Staubli VAL3: decode.pgx

public program decode(num& x_nStatus (dimensions=1), num& x_nDWordBody[] (dimensions=2))
  local num l_nBodyDWordLen
  local num i
begin
  // x_nStatus
  // -1 - unsuccessful
  // 0 - successful
  x_nStatus=-1
  l_nBodyDWordLen=34
  if size(x_nDWordBody,1)!=l_nBodyDWordLen or size(x_nDWordBody,2)!=4
    put("Size of the param is: "+toString("",size(x_nDWordBody,1)))
    putln("x"+toString("",size(x_nDWordBody,2)))
    return
  endIf
  x_nStatus=0
  call decodeSharedInt(x_nStatus,body.robotId,x_nDWordBody,0)
  call decodeSharedInt(x_nStatus,body.sequence,x_nDWordBody,1)
  call decodeSharedInt(x_nStatus,body.validFields,x_nDWordBody,2)
  call decodeShareReal(x_nStatus,body.time,x_nDWordBody,3)
  call decodeJointData(x_nStatus,body.positions,x_nDWordBody,4)
  call decodeJointData(x_nStatus,body.velocities,x_nDWordBody,14)
  call decodeJointData(x_nStatus,body.accelerations,x_nDWordBody,24)
end
